FUNCTION "LGF_CompareVariant" : Bool
TITLE = LGF_CompareVariant
{ S7_Optimized_Access := 'TRUE' }
AUTHOR : Siemens_Digital_Industry
FAMILY : LGF
NAME : LGF_CompareVariant
//The function compares two structured actual parameters (array, PLC data type) and outputs whether they are of the same type and have the same values.
//
//Compare arrays or plc datatypes and their values up to a max lengh of 200 Bytes of the connected variables. If at least one value of an element is not identical --> set function result = false
//
//Restrictions:
//The attached structure must not include Strings
//The attached structure can not exceed 200 bytes, because of the internal buffer size
   VAR_OUTPUT
      error : Bool;   // FALSE: No error / TRUE: An error occurred during the execution of the FB
      status : Word;   // 16#0000-16#7FFF: Status of the FB / 16#8000-16#FFFF: Error identification (see following Table)
      subFunctionStatus : Word;   // Status or return value of called FB's, FC's and system blocks
   END_VAR

   VAR_IN_OUT
      variableA : Variant;   // First comparison variable with any data type
      variableB : Variant;   // Second comparison variable with any data type
   END_VAR

   VAR_TEMP
      tempVariableASize : DInt;   // Temp store length of serialized structur of `variableA`
      tempVariableBSize : DInt;   // Temp store length of serialized of `variableB`
      tempindex : DInt;   // Temp index to loop trough serialzed byte arrays for comparision
      tempVariableAToBytes : Array[0..#MAX_LENGTH] of Byte;   // Temp store for serialized structure  of `variableA`
      tempVariableBToBytes : Array[0..#MAX_LENGTH] of Byte;   // Temp store for serialized of `variableB`
      tempSerializeRet : Word;   // Temp `serialize` result - Errorcode >= 16#8000 if function fails
   END_VAR

   VAR CONSTANT
      STATUS_NO_ERROR : Word := 16#0000;   // Execution finished without errors
      ERR_INPUT_TYPES_MUST_MATCH : Word := 16#8201;   // Error, the input types must match, e.g. STRUCT
      ERR_INPUT_TYPES_LENGTH_NOT_EQUAL : Word := 16#8202;   // Error, the input types have different lengths after serialization, `subFunctionStatus` provides an indicator of the different size
      ERR_SERIALIZE_VARIABLE_A : Word := 16#8601;   // Error occured while serialize variableA into Bytearray - see `subFunctionStatus` for detailed information
      ERR_SERIALIZE_VARIABLE_B : Word := 16#8602;   // Error occured while serialize variableB into Bytearray - see `subFunctionStatus` for detailed information
      MAX_LENGTH : Int := 200;   // Max. length of PLC data structur in Bytes, defines the internal buffer size
   END_VAR


BEGIN
	REGION BLOCK INFO HEADER
	  //===============================================================================
	  // SIEMENS AG / (c)Copyright 2019
	  //-------------------------------------------------------------------------------
	  // Title:            LGF_CompareVariant
	  // Comment/Function: Compare arrays or plc datatypes and their values
	  //                   up to a max lengh of 200 Bytes of the connected variables.
	  //                   If at least one value of an element is not identical -->
	  //                   set function result = false
	  // Library/Family:   LGF (Library General Functions)
	  // Author:           Siemens Digital Industry
	  // Tested with:      CPU1212C DC/DC/DC FW:V4.2
	  // Engineering:      TIA Portal V15.1
	  // Restrictions:     The attached structure must not include Strings
	  //                   The attached structure can not exceed 200 bytes,
	  //                   because of the internal buffer size
	  //                   --> extend: cut from type, adjust "MAX_LENGHT" constant
	  //                   ENO disabled - error handling done with error and status
	  // Requirements:     PLC (S7-1200 / S7-1500)
	  //-------------------------------------------------------------------------------
	  // Change log table:
	  // Version  | Date       | Expert in charge       | Changes applied
	  // 01.00.00 03.09.2015  Siemens Industry Online Support
	  //                      First released version
	  // 01.00.01 11.02.2015  Siemens Industry Online Support
	  //                      Bug fix
	  // 01.00.02 02.01.2017  Siemens Industry Online Support
	  //                      Upgrade: TIA V14 Update 1
	  // 01.00.03 17.08.2018  Siemens Industry Online Support
	  //                      Upgrade: TIA V15 Update 2
	  // 01.00.04 23.11.2018  Siemens Industry Online Support
	  //                      Upgrade: TIA V15.1
	  // 01.00.05 03.06.2019  Simatic Systems Support
	  //                      Refactoring and performance improvment
	  //                      Change error handling to status and subFctStatus
	  //                      update serialize instruction
	  //                      add eno handling
	  // 03.00.00 23.04.2020  Simatic Systems Support
	  //                      Set version to V3.0.0, harmonize the version of the whole library
	  // 03.00.01 19.01.2020  Simatic Systems Support
	  //                      Insert documentation
	  //===============================================================================
	END_REGION BLOCK INFO HEADER

	REGION DESCRIPTION
	  (/*
	NOTE
	:    The status of called commands is output in `subFunctionStatus`. In this case, the output value in `status` indicates which command caused the error. In this case, refer to the TIA Portal Online Help section for information on the respective commands.

	---

	This block compares two (structured) actual parameters and shows whether they equate to the same value.

	Note
	:    The following differences cannot be detected with the comparison method (byte level):
	* Variables of the data type `Struct` cannot be compared.
	* For strings, there may be differences in the range between the actual length and the maximum length.
	* With `REAL` numbers in the structure, a disparity can also be displayed for "same" variables.
	* Variables of the type `ARRAY of BOOL` cannot be checked for equality with the function, because the command used, `CountOfElements`, also counts the filling elements (e.g. 8 is returned with an `ARRAY[0..1] of BOOL`).
	*/)
	END_REGION DESCRIPTION

	REGION Initialisation
	  // init temporary variables
	  #tempVariableASize := 0;
	  #tempVariableBSize := 0;
	  #tempindex := 0;

	  // Set "No current job" #status
	  #error := FALSE;
	  #status := #STATUS_NO_ERROR;
	  #subFunctionStatus := #STATUS_NO_ERROR;

	  // Initialisation of function result
	  #LGF_CompareVariant := FALSE;
	END_REGION Initialisation

	REGION Processing

	  REGION Check input types
	    // Check if the datatypes of the connected tags are identical
	    IF TypeOf(#variableA) <> TypeOf(#variableB) THEN
	      #error := TRUE;
	      #status := #ERR_INPUT_TYPES_MUST_MATCH;
	      #subFunctionStatus := #STATUS_NO_ERROR;
	      // no error handling needed
	      ENO := TRUE;
	      RETURN; // Finish function if conversion fails
	    END_IF;
	  END_REGION

	  REGION Serialize Input Variable A
	    // convert variableA Values to serialised binary array of byte
	    #tempSerializeRet := INT_TO_WORD(
	                                     Serialize(SRC_VARIABLE := #variableA,
	                                               DEST_ARRAY => #tempVariableAToBytes,
	                                               POS := #tempVariableASize)
	    );

	    // Check return value of SERIALIZE
	    // if not zero - error happend, write error codes and end/leave function
	    IF #tempSerializeRet <> #STATUS_NO_ERROR THEN
	      #error := TRUE;
	      #status := #ERR_SERIALIZE_VARIABLE_A;
	      #subFunctionStatus := #tempSerializeRet;
	      // no error handling needed
	      ENO := TRUE;
	      RETURN; // Finish function if conversion fails
	    END_IF;
	  END_REGION

	  REGION Serialize Input Variable A
	    // convert variableB Values to serialised binary array of byte
	    #tempSerializeRet := INT_TO_WORD(
	                                     Serialize(SRC_VARIABLE := #variableB,
	                                               DEST_ARRAY => #tempVariableBToBytes,
	                                               POS := #tempVariableBSize)
	    );

	    // Check return value of SERIALIZE
	    // if not zero - error happend, write error codes and end/leave function
	    IF #tempSerializeRet <> #STATUS_NO_ERROR THEN
	      #error := TRUE;
	      #status := #ERR_SERIALIZE_VARIABLE_B;
	      #subFunctionStatus := #tempSerializeRet;
	      // no error handling needed
	      ENO := TRUE;
	      RETURN; // Finish function if conversion fails
	    END_IF;
	  END_REGION

	  REGION Check if serialized sizes are equal
	    // Compare size of both variables
	    IF #tempVariableASize <> #tempVariableBSize THEN
	      #error := TRUE;
	      #status := #ERR_INPUT_TYPES_LENGTH_NOT_EQUAL;
	      #subFunctionStatus := DINT_TO_WORD(#tempVariableASize - #tempVariableBSize);
	      // no error handling needed
	      ENO := TRUE;
	      RETURN; // Finish function if conversion fails
	    END_IF;
	  END_REGION

	  REGION Compare
	    // Compare values of temp. array elements of bytes
	    WHILE #tempindex < #tempVariableASize DO

	      // Compare bytes till difference detected
	      IF #tempVariableAToBytes[#tempindex] = #tempVariableBToBytes[#tempindex] THEN
	        // if equal increment index
	        #tempindex += 1; // Or end of array reached
	      ELSE
	        // if values diffrent (content missmatch) --> exit loop
	        EXIT;
	      END_IF;
	    END_WHILE;

	  END_REGION
	END_REGION Processing

	REGION Output
	  // Assign function result - if index is equal to size = TRUE
	  #LGF_CompareVariant := (#tempindex = #tempVariableASize);

	  // ENO is not used, forced to TRUE
	  ENO := TRUE;
	END_REGION

END_FUNCTION

